FUNCTION_BLOCK MUL_REAL (* IEC 61131-3 REAL Multiplication *)
  (* Standard: 61131-3 *)
  (* Version 0.0, 2004-12-15, JHC, Rockwell Automation, Converted from SRC format. *)
  (* Compiler header: package fb.rt.plc.math; *)
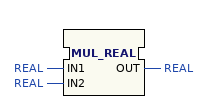
  VAR_INPUT
    IN1 : REAL; (* Multiplicand *)
    IN2 : REAL; (* Multiplier *)
  END_VAR
  VAR_OUTPUT
    OUT : REAL; (* Product *)
  END_VAR
END_FUNCTION_BLOCK
